// TIA Portal project "MojProjekat" (V16)

(* hardware
DEVICE "S7300/ET200M station_1"  S7-300 station
   slot 0: "Rail_0"  Rail  6ES7 390-1***0-0AA0
   slot 1: "PS 305 2A Outdoor_1"  PS 305 2A Outdoor  6ES7 305-1BA80-0AA0
   slot 2: "PLC_1"  CPU 315-2 PN/DP  6ES7 315-2EH14-0AB0  V3.2
      slot 2: "PROFINET interface_1"  PN-IO
         slot 1: "Port_1"  Port
         slot 2: "Port_2"  Port
   slot 4: "DI 32x24VDC_1"  DI32 x 24VDC  6ES7 321-1BL00-0AA0
   slot 5: "DO 32x24VDC/0.5A_1"  DO32 x 24VDC / 0.5A  6ES7 322-1BL00-0AA0
   slot 6: "DI 16/DO 16x24VDC/0.5A_1"  DI16/DO16 x 24V / 0.5A  6ES7 323-1BL00-0AA0
   slot 7: "AI 2x12BIT_1"  AI2 x 12 bits  6ES7 331-7KB02-0AB0
*)

// ===== PLC "PLC_1"  CPU 315-2 PN/DP =====

VAR_GLOBAL   // PLC tag table "Default tag table"
   "Tag_1" AT %M500.0 : Bool;
   "Tag_2" AT %M500.1 : Bool;
   "Tag_3" AT %C18 : Counter;
   "Tag_4" AT %M77.0 : Bool;
END_VAR

VAR_GLOBAL   // PLC tag table "STEP7 classic symbols"
   "M_Bays_occup_HMI" AT %M33.0 : Bool;   // all Bays 1 to 3 occupied
   "M_Ackn_Fault_HMI" AT %M31.0 : Bool;   // Memory bit, acknowledge conveyor fault (TP177)
   "M_M/A_Accept_HMI" AT %M30.5 : Bool;   // Memory bit, confirm operating mode (TP177)
   "M_M/A_ModeSelect_HMI" AT %M30.4 : Bool;   // Memory bit Operating Mode Preselect: '0'=MANUAL, '1'=AUTO (TP177)
   "M_Conv_Jog_LEFT_HMI" AT %M30.3 : Bool;   // Memory bit Jog Conveyor LEFT (TP177)
   "M_Conv_Jog_RIGHT_HMI" AT %M30.2 : Bool;   // Memory bit Jog Conveyor RIGHT (TP177)
   "M_System_OFF_HMI" AT %M30.1 : Bool;   // Memory bit System OFF (TP177)
   "M_System_ON_HMI" AT %M30.0 : Bool;   // Memory bit System ON (TP177)
   "M_Aux_Count" AT %M19.0 : Bool;   // Edge auxiliary memory bit Light barrier
   "M_Aux_Auto" AT %M18.0 : Bool;   // Auxiliary memory bit Edge AUTO on
   "T_M/A_Accept" AT %I0.5 : Bool;   // Momentary contact, confirm operating mode
   "S_M/A_ModeSelect" AT %I0.4 : Bool;   // Switch - Operating Mode Preselect: '0'=MANUAL, '1'=AUTO
   "T_Jog_LEFT" AT %I0.3 : Bool;   // Jog conveyor LEFT, momentary contact
   "T_Jog_RIGHT" AT %I0.2 : Bool;   // Jog conveyor RIGHT, momentary contact
   "T_System_OFF" AT %I0.1 : Bool;   // Momentary contact System OFF (NC contact)
   "T_System_ON" AT %I0.0 : Bool;   // Momentary contact System ON
   "MW_Messages" AT %MW32 : Word;   // Trigger variable for WinCC flexible - Messages
   "MW_SETP" AT %MW22 : Int;   // Memory word, SETPOINT quantity of parts to be transp.
   "MW_ACT" AT %MW20 : Int;   // Memory word, ACTUAL quantity of transported parts
   "MD_Slave_Recovery" AT %MD96 : Time_Of_Day;   // Time when slave recovered
   "MD_Slave_Failure" AT %MD92 : Time_Of_Day;   // Time when DP slave failed
   "MD_Slave_Downtime" AT %MD88 : Time;   // Down time of slave
   "MB_Step_mem_bit" AT %MB100 : Byte;   // Memory byte with step memory bit
   "L_Bay-LB" AT %Q8.4 : Bool;   // Indicator light Light barrier bay
   "L_Bay3" AT %Q8.3 : Bool;   // Indicator light Bay 3
   "L_Bay2" AT %Q8.2 : Bool;   // Indicator light Bay 2
   "BAY2" AT %I8.6 : Bool;   // Proximity sensor Bay 2
   "BAY1" AT %I8.5 : Bool;   // Proximity sensor Bay 1
   "T_Bay-LB" AT %I8.4 : Bool;   // Momentary contact Light barrier bay
   "T_Bay3" AT %I8.3 : Bool;   // Momentary contact Bay 3
   "T_Bay2" AT %I8.2 : Bool;   // Momentary contact Bay 2
   "T_Bay1" AT %I8.1 : Bool;   // Momentary contact Bay 1
   "LB" AT %I8.0 : Bool;   // Light barrier
   "S_Fault3" AT %I1.3 : Bool;   // Simulate Fault 3, 0=OFF/1=ON
   "S_Fault2" AT %I1.2 : Bool;   // Simulate Fault 2, 0=OFF/1=ON
   "S_Fault1" AT %I1.1 : Bool;   // Simulate Fault 1, 0=OFF/1=ON
   "QW_Setp_G120" AT %QW44 : Word;   // Setpoint speed for G120
   "QW_Control_G120" AT %QW42 : Word;   // Control word for G120
   "QW_DigDisp" AT %QW6 : Word;   // BCD digital display
   "QB_Simulator-LED" AT %QB5 : Byte;   // lower Simulator LEDs
   "Horn" AT %Q8.7 : Bool;   // Horn
   "K_Conv_LEFT" AT %Q8.6 : Bool;   // Run conveyor LEFT
   "K_Conv_RIGHT" AT %Q8.5 : Bool;   // Run conveyor RIGHT
   "M_Aux_Fault2" AT %M17.4 : Bool;   // Edge auxiliary memory bit Fault 2
   "M_Fault2" AT %M17.3 : Bool;   // Memory bit for storing Fault 2
   "M_Aux_Fault1" AT %M17.2 : Bool;   // Edge auxiliary memory bit Fault 1
   "M_Fault1" AT %M17.1 : Bool;   // Memory bit for storing Fault 1
   "M_Conv_Fault" AT %M17.0 : Bool;   // Memory bit Conveyor fault
   "MB_SlaveAddress" AT %MB87 : Byte;   // DP address of failed slave
   "M_InitialState" AT %M101.1 : Bool;   // Memory bit, production line in initial state
   "M_Edge_Aux" AT %M101.0 : Bool;   // Auxiliary memory bit Edge detection AUTO on
   "M_S6_Final_Check" AT %M100.6 : Bool;   // Step 6: Final check
   "M_S5_3->LB" AT %M100.5 : Bool;   // Step 5: Transport Bay 3 -> Light barrier bay
   "OD_Conv_Monitoring" AT %T17 : Timer;   // Timer, Conveyor monitoring in Auto mode
   "OD_Milling" AT %T4 : Timer;   // Timer for simulating the milling
   "OD_Drilling" AT %T2 : Timer;   // Timer for simulating the drilling
   "M_S4_Mill" AT %M100.4 : Bool;   // Step 4: Mill
   "M_S3_2->3" AT %M100.3 : Bool;   // Step 3: Transport from Bay 2 -> 3
   "M_S2_Drill" AT %M100.2 : Bool;   // Step 2: Drill at Bay 2
   "M_S1_1->2" AT %M100.1 : Bool;   // Step 1: Transport from Bay 1 > 2
   "M_S0_Init" AT %M100.0 : Bool;   // Memory bit InitialStep
   "M_SlaveFailure" AT %M86.0 : Bool;   // Memory bit DP Slave has failed
   "M_G120_Jog_LEFT_HMI" AT %M40.3 : Bool;   // Memory bit G120 Jog LEFT (TP177)
   "M_G120_Jog_RIGHT_HMI" AT %M40.2 : Bool;   // Memory bit G120 Jog RIGHT (TP177)
   "M_G120_On_HMI" AT %M40.0 : Bool;   // Switch On Memory bit G120 (TP177)
   "M_Weight_ok" AT %M35.0 : Bool;   // is equal to 1 when weight ok
   "IW_State_G120" AT %IW42 : Word;   // State word of G120
   "IW_Thumbw" AT %IW2 : Word;   // BCD thumbwheel
   "BAY3" AT %I8.7 : Bool;   // Proximity sensor Bay 3
   "L_Bay1" AT %Q8.1 : Bool;   // Indicator light Bay 1
   "L_S6_Final_Check" AT %Q5.6 : Bool;   // Indicator light Final check at LB bay
   "L_S5_3->LB" AT %Q5.5 : Bool;   // Indicator light Transport Bay 3 -> Light barrier bay
   "L_S4_Mill" AT %Q5.4 : Bool;   // Indicator light Milling at Bay 3
   "L_Fault3" AT %Q5.3 : Bool;   // Indicator light Fault 3
   "L_Fault2" AT %Q5.2 : Bool;   // Indicator light Fault 2
   "L_Fault1" AT %Q5.1 : Bool;   // Indicator light Fault 1
   "L_Conv_Fault" AT %Q5.0 : Bool;   // Indicator light Conveyor fault
   "L_Restart_aut" AT %Q4.6 : Bool;   // Indicator light for automatic warm restart
   "L_Restart_man" AT %Q4.5 : Bool;   // Indicator light for manual warm restart
   "M_Aux_Man_ON" AT %M15.2 : Bool;   // Edge auxiliary memory bit Manual mode ON
   "M_Aux_System_ON" AT %M15.1 : Bool;   // Edge auxiliary memory bit System ON
   "M_Bay3_occup" AT %M14.3 : Bool;   // Memory bit Bay 3 occupied
   "M_Bay2_occup" AT %M14.2 : Bool;   // Memory bit Bay 2 occupied
   "M_Bay1_occup" AT %M14.1 : Bool;   // Memory bit Bay 1 occupied
   "M_Aux_Left" AT %M14.0 : Bool;   // Aux. memory bit Edge Conv LEFT Stop
   "M_Flash_1Hz" AT %M10.5 : Bool;   // Memory bit - flashing frequency 1Hz
   "M_Flash_2Hz" AT %M10.3 : Bool;   // Memory bit - flashing frequency 2 Hz
   "IW_Act_G120" AT %IW44 : Word;   // Actual speed of G120
   "M_Conv_Fault_HMI" AT %M33.1 : Bool;   // Memory bit Conveyor fault
   "C_Conv_Fault" AT %C17 : Counter;   // Counter Conveyor faults
   "C_Bay3" AT %C3 : Counter;   // Counter Bay 3
   "C_Bay2" AT %C2 : Counter;   // Counter Bay 2
   "C_Bay1" AT %C1 : Counter;   // Counter Bay 1
   "L_AUTO" AT %Q4.3 : Bool;   // Indicator light Automatic mode
   "L_MAN" AT %Q4.2 : Bool;   // Indicator light MAN mode
   "L_SYSTEM" AT %Q4.1 : Bool;   // Indicator light System ON
   "T_Ackn_Fault" AT %I1.0 : Bool;   // Momentary contact Fault acknowledgement
   "T_Ackn_WarmRestart" AT %I0.7 : Bool;   // Momentary contact to acknowledge warm restart display
   "S_Weight/Quantity" AT %I0.6 : Bool;   // 0 = Display quantity, 1 = Display weight
   "M_Auto_LEFT" AT %M16.6 : Bool;   // Memory bit Conveyor AUTO LEFT
   "M_Auto_RIGHT" AT %M16.4 : Bool;   // Memory bit Conveyor AUTO RIGHT
   "M_Jog_LEFT" AT %M16.3 : Bool;   // Memory bit Jog conveyor LEFT
   "M_Jog_RIGHT" AT %M16.2 : Bool;   // Memory bit Jog conveyor RIGHT
   "M_Aux_LB" AT %M16.0 : Bool;   // Edge auxiliary memory bit Light barrier
   "M_Aux_C17" AT %M15.7 : Bool;   // Edge auxiliary memory bit Counter-Conveyor faults
   "M_Aux_Auto_ON" AT %M15.3 : Bool;   // Edge auxiliary memory bit Auto mode ON
   "M_Setpoint_reached_HMI" AT %M33.2 : Bool;   // Memory bit Setpoint reached
   "L_Weight_invalid" AT %Q4.0 : Bool;   // Indicator light - weight invalid
   "P_PIW_AI2" AT %IW306 : Int;   // Simulator-Poti for presetting G120 speed
   "P_PIW_AI1" AT %IW304 : Int;   // Simulator-Poti for presetting weight
   "MW_Weight" AT %MW36 : Int;   // Memory word with current weight
END_VAR

FUNCTION "FC_14" : Void   // FC14, LAD
{ S7_Optimized_Access := 'FALSE' }
VERSION : 0.1
BEGIN

REGION Network 1: Indicator light Bay 1
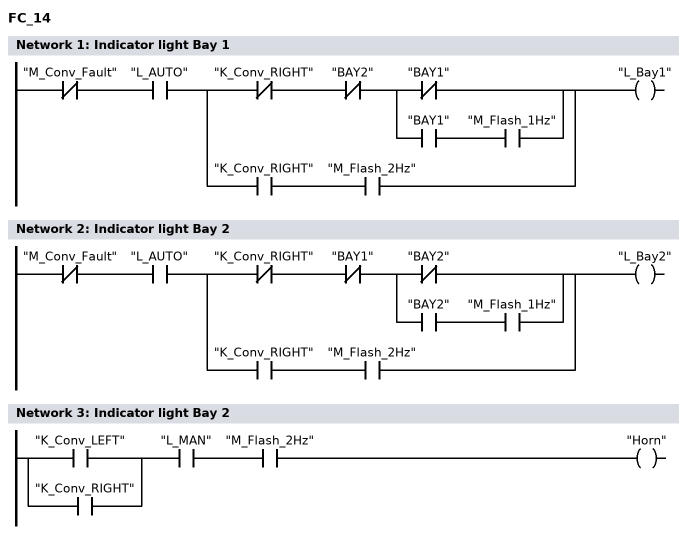
   RUNG wire#powerrail
      I_Contact( "M_Conv_Fault" )
      Contact( "L_AUTO" )
      wire#w1
      I_Contact( "K_Conv_RIGHT" )
      I_Contact( "BAY2" )
      wire#w2
      I_Contact( "BAY1" )
      wire#w3
      Coil( "L_Bay1" )
   END_RUNG
   RUNG wire#w2
      Contact( "BAY1" )
      Contact( "M_Flash_1Hz" )
   END_RUNG wire#w3
   RUNG wire#w1
      Contact( "K_Conv_RIGHT" )
      Contact( "M_Flash_2Hz" )
   END_RUNG wire#w3
   // the same network as SCL:
   "L_Bay1" := NOT "M_Conv_Fault" AND "L_AUTO" AND ((NOT "K_Conv_RIGHT" AND NOT "BAY2" AND (NOT "BAY1" OR ("BAY1" AND "M_Flash_1Hz"))) OR ("K_Conv_RIGHT" AND "M_Flash_2Hz"));
END_REGION

REGION Network 2: Indicator light Bay 2
   RUNG wire#powerrail
      I_Contact( "M_Conv_Fault" )
      Contact( "L_AUTO" )
      wire#w1
      I_Contact( "K_Conv_RIGHT" )
      I_Contact( "BAY1" )
      wire#w2
      I_Contact( "BAY2" )
      wire#w3
      Coil( "L_Bay2" )
   END_RUNG
   RUNG wire#w2
      Contact( "BAY2" )
      Contact( "M_Flash_1Hz" )
   END_RUNG wire#w3
   RUNG wire#w1
      Contact( "K_Conv_RIGHT" )
      Contact( "M_Flash_2Hz" )
   END_RUNG wire#w3
   // the same network as SCL:
   "L_Bay2" := NOT "M_Conv_Fault" AND "L_AUTO" AND ((NOT "K_Conv_RIGHT" AND NOT "BAY1" AND (NOT "BAY2" OR ("BAY2" AND "M_Flash_1Hz"))) OR ("K_Conv_RIGHT" AND "M_Flash_2Hz"));
END_REGION

REGION Network 3: Indicator light Bay 2
   RUNG wire#powerrail
      Contact( "K_Conv_LEFT" )
      wire#w1
      Contact( "L_MAN" )
      Contact( "M_Flash_2Hz" )
      Coil( "Horn" )
   END_RUNG
   RUNG wire#powerrail
      Contact( "K_Conv_RIGHT" )
   END_RUNG wire#w1
   // the same network as SCL:
   "Horn" := ("K_Conv_LEFT" OR "K_Conv_RIGHT") AND "L_MAN" AND "M_Flash_2Hz";
END_REGION
END_FUNCTION

FUNCTION "FC_Mode" : Void   // FC15, LAD
{ S7_Optimized_Access := 'FALSE' }
VERSION : 0.1
   VAR_TEMP   // added for the SCL form of the ladder/FBD networks
      _w1 : Bool;
   END_VAR
BEGIN

REGION Network 1
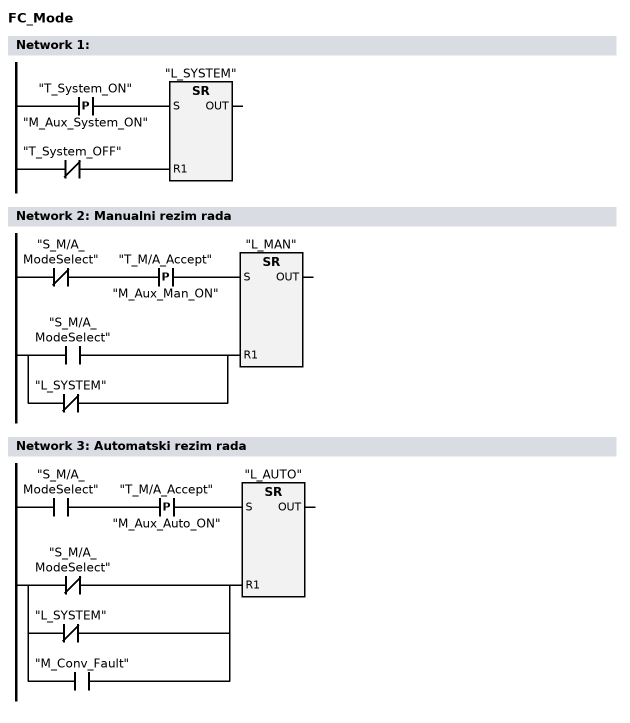
   RUNG wire#powerrail
      P_Contact(operand := "T_System_ON", bit := "M_Aux_System_ON")
      S_SR(operand := "L_SYSTEM", r1 := wire#w1)
   END_RUNG
   RUNG wire#powerrail
      I_Contact( "T_System_OFF" )
   END_RUNG wire#w1
   // the same network as SCL:
   #_w1 := "T_System_ON" AND NOT "M_Aux_System_ON";   // rising edge of "T_System_ON"
   "M_Aux_System_ON" := "T_System_ON";
   IF #_w1 THEN
       "L_SYSTEM" := TRUE;   // SR flip-flop
   END_IF;
   IF NOT "T_System_OFF" THEN "L_SYSTEM" := FALSE; END_IF;
END_REGION

REGION Network 2: Manualni rezim rada
   RUNG wire#powerrail
      I_Contact( "S_M/A_ModeSelect" )
      P_Contact(operand := "T_M/A_Accept", bit := "M_Aux_Man_ON")
      S_SR(operand := "L_MAN", r1 := wire#w1)
   END_RUNG
   RUNG wire#powerrail
      Contact( "S_M/A_ModeSelect" )
   END_RUNG wire#w1
   RUNG wire#powerrail
      I_Contact( "L_SYSTEM" )
   END_RUNG wire#w1
   // the same network as SCL:
   #_w1 := NOT "S_M/A_ModeSelect" AND "T_M/A_Accept" AND NOT "M_Aux_Man_ON";   // rising edge of "T_M/A_Accept"
   "M_Aux_Man_ON" := "T_M/A_Accept";
   IF #_w1 THEN
       "L_MAN" := TRUE;   // SR flip-flop
   END_IF;
   IF "S_M/A_ModeSelect" OR NOT "L_SYSTEM" THEN "L_MAN" := FALSE; END_IF;
END_REGION

REGION Network 3: Automatski rezim rada
   RUNG wire#powerrail
      Contact( "S_M/A_ModeSelect" )
      P_Contact(operand := "T_M/A_Accept", bit := "M_Aux_Auto_ON")
      S_SR(operand := "L_AUTO", r1 := wire#w1)
   END_RUNG
   RUNG wire#powerrail
      I_Contact( "S_M/A_ModeSelect" )
   END_RUNG wire#w1
   RUNG wire#powerrail
      I_Contact( "L_SYSTEM" )
   END_RUNG wire#w1
   RUNG wire#powerrail
      Contact( "M_Conv_Fault" )
   END_RUNG wire#w1
   // the same network as SCL:
   #_w1 := "S_M/A_ModeSelect" AND "T_M/A_Accept" AND NOT "M_Aux_Auto_ON";   // rising edge of "T_M/A_Accept"
   "M_Aux_Auto_ON" := "T_M/A_Accept";
   IF #_w1 THEN
       "L_AUTO" := TRUE;   // SR flip-flop
   END_IF;
   IF NOT "S_M/A_ModeSelect" OR NOT "L_SYSTEM" OR "M_Conv_Fault" THEN "L_AUTO" := FALSE; END_IF;
END_REGION
END_FUNCTION

FUNCTION "FC_Conveyor" : Void   // FC16, LAD
{ S7_Optimized_Access := 'FALSE' }
VERSION : 0.1
   VAR_TEMP   // added for the SCL form of the ladder/FBD networks
      _w1 : Bool;
   END_VAR
BEGIN

REGION Network 1: Run conveyor RIGHT
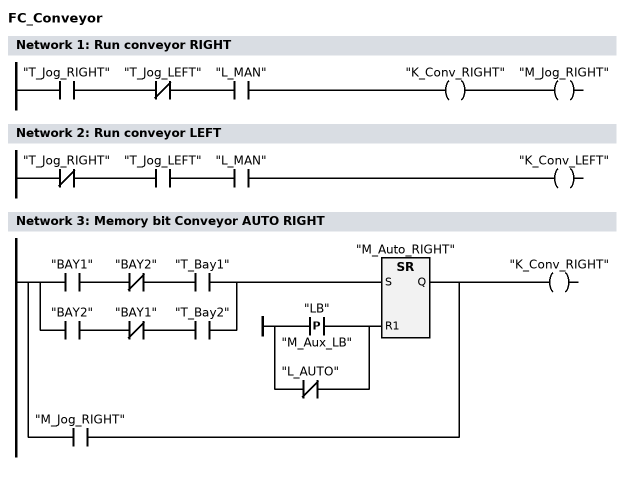
   RUNG wire#powerrail
      Contact( "T_Jog_RIGHT" )
      I_Contact( "T_Jog_LEFT" )
      Contact( "L_MAN" )
      Coil( "K_Conv_RIGHT" )
      Coil( "M_Jog_RIGHT" )
   END_RUNG
   // the same network as SCL:
   "K_Conv_RIGHT" := "T_Jog_RIGHT" AND NOT "T_Jog_LEFT" AND "L_MAN";
   "M_Jog_RIGHT" := "K_Conv_RIGHT";
END_REGION

REGION Network 2: Run conveyor LEFT
   RUNG wire#powerrail
      I_Contact( "T_Jog_RIGHT" )
      Contact( "T_Jog_LEFT" )
      Contact( "L_MAN" )
      Coil( "K_Conv_LEFT" )
   END_RUNG
   // the same network as SCL:
   "K_Conv_LEFT" := NOT "T_Jog_RIGHT" AND "T_Jog_LEFT" AND "L_MAN";
END_REGION

REGION Network 3: Memory bit Conveyor AUTO RIGHT
   RUNG wire#powerrail
      Contact( "BAY1" )
      I_Contact( "BAY2" )
      Contact( "T_Bay1" )
      wire#w1
      S_SR(operand := "M_Auto_RIGHT", r1 := wire#w2)
      wire#w3
      Coil( "K_Conv_RIGHT" )
   END_RUNG
   RUNG wire#powerrail
      Contact( "BAY2" )
      I_Contact( "BAY1" )
      Contact( "T_Bay2" )
   END_RUNG wire#w1
   RUNG wire#powerrail
      P_Contact(operand := "LB", bit := "M_Aux_LB")
   END_RUNG wire#w2
   RUNG wire#powerrail
      I_Contact( "L_AUTO" )
   END_RUNG wire#w2
   RUNG wire#powerrail
      Contact( "M_Jog_RIGHT" )
   END_RUNG wire#w3
   // the same network as SCL:
   #_w1 := "LB" AND NOT "M_Aux_LB";   // rising edge of "LB"
   "M_Aux_LB" := "LB";
   IF ("BAY1" AND NOT "BAY2" AND "T_Bay1") OR ("BAY2" AND NOT "BAY1" AND "T_Bay2") THEN
       "M_Auto_RIGHT" := TRUE;   // SR flip-flop
   END_IF;
   IF #_w1 OR NOT "L_AUTO" THEN "M_Auto_RIGHT" := FALSE; END_IF;
   "K_Conv_RIGHT" := "M_Auto_RIGHT" OR "M_Jog_RIGHT";
END_REGION
END_FUNCTION

FUNCTION "FC_FAULT" : Void   // FC17, LAD
{ S7_Optimized_Access := 'FALSE' }
VERSION : 0.1
   VAR_TEMP   // added for the SCL form of the ladder/FBD networks
      _w1 : Bool;
      _s5time1 : S5Time;
   END_VAR
BEGIN

REGION Network 1: Indicator light Conveyor fault
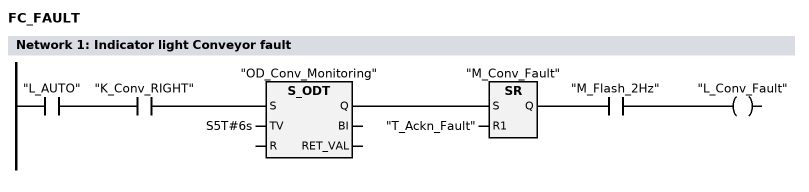
   RUNG wire#powerrail
      Contact( "L_AUTO" )
      Contact( "K_Conv_RIGHT" )
      S_ODT(T_NO := "OD_Conv_Monitoring", TV := S5T#6s, R :=, BI =>, RET_VAL =>)
      S_SR(operand := "M_Conv_Fault", r1 := "T_Ackn_Fault")
      Contact( "M_Flash_2Hz" )
      Coil( "L_Conv_Fault" )
   END_RUNG
   // the same network as SCL:
   #_s5time1 := S_ODT(T_NO := "OD_Conv_Monitoring", S := "L_AUTO" AND "K_Conv_RIGHT", TV := S5T#6s, Q => #_w1);
   IF #_w1 THEN
       "M_Conv_Fault" := TRUE;   // SR flip-flop
   END_IF;
   IF "T_Ackn_Fault" THEN "M_Conv_Fault" := FALSE; END_IF;
   "L_Conv_Fault" := "M_Conv_Fault" AND "M_Flash_2Hz";
END_REGION
END_FUNCTION

FUNCTION "FC_Count" : Void   // FC18, LAD
{ S7_Optimized_Access := 'FALSE' }
VERSION : 0.1
   VAR_TEMP   // added for the SCL form of the ladder/FBD networks
      _w1 : Bool;
   END_VAR
BEGIN

REGION Network 1
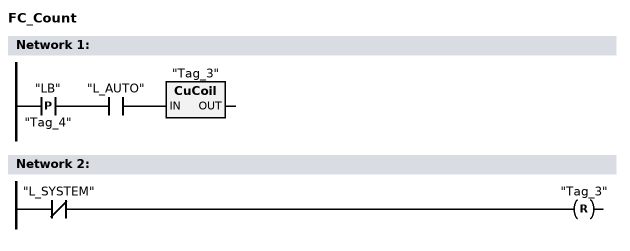
   // no SCL statement known for CuCoil: written as a call
   #_w1 := "LB" AND NOT "Tag_4";   // rising edge of "LB"
   "Tag_4" := "LB";
   CuCoil(in := #_w1 AND "L_AUTO", operand := "Tag_3");
END_REGION

REGION Network 2
   RUNG wire#powerrail
      I_Contact( "L_SYSTEM" )
      R_Coil( "Tag_3" )
   END_RUNG
   // the same network as SCL:
   IF NOT "L_SYSTEM" THEN "Tag_3" := FALSE; END_IF;
END_REGION
END_FUNCTION

ORGANIZATION_BLOCK "Main"   // OB1, LAD
TITLE = "Main Program Sweep (Cycle)"
{ S7_Optimized_Access := 'FALSE' }
VERSION : 0.1
   VAR_TEMP
      OB1_EV_CLASS : Byte;   // Bits 0-3 = 1 (Coming event), Bits 4-7 = 1 (Event class 1)
      OB1_SCAN_1 : Byte;   // 1 (Cold restart scan 1 of OB 1), 3 (Scan 2-n of OB 1)
      OB1_PRIORITY : Byte;   // Priority of OB Execution
      OB1_OB_NUMBR : Byte;   // 1 (Organization block 1, OB1)
      OB1_RESERVED_1 : Byte;   // Reserved for system
      OB1_RESERVED_2 : Byte;   // Reserved for system
      OB1_PREV_CYCLE : Int;   // Cycle time of previous OB1 scan (milliseconds)
      OB1_MIN_CYCLE : Int;   // Minimum cycle time of OB1 (milliseconds)
      OB1_MAX_CYCLE : Int;   // Maximum cycle time of OB1 (milliseconds)
      OB1_DATE_TIME : Date_And_Time;   // Date and time OB1 started
   END_VAR
BEGIN

REGION Network 1: Operation Modes
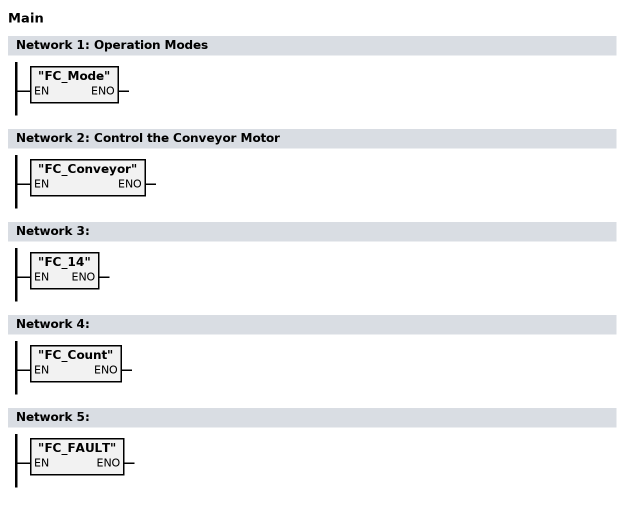
   RUNG wire#powerrail
      "FC_Mode"()
   END_RUNG
   // the same network as SCL:
   "FC_Mode"();
END_REGION

REGION Network 2: Control the Conveyor Motor
   RUNG wire#powerrail
      "FC_Conveyor"()
   END_RUNG
   // the same network as SCL:
   "FC_Conveyor"();
END_REGION

REGION Network 3
   RUNG wire#powerrail
      "FC_14"()
   END_RUNG
   // the same network as SCL:
   "FC_14"();
END_REGION

REGION Network 4
   RUNG wire#powerrail
      "FC_Count"()
   END_RUNG
   // the same network as SCL:
   "FC_Count"();
END_REGION

REGION Network 5
   RUNG wire#powerrail
      "FC_FAULT"()
   END_RUNG
   // the same network as SCL:
   "FC_FAULT"();
END_REGION
END_ORGANIZATION_BLOCK